// TIA Portal V16 export
// export: Created 2021-11-12T13:32:10.6511653Z, ExportSetting WithDefaults, DisplayName Totally Integrated Automation Portal, DisplayVersion V16 Update 3, DisplayName TIA Portal Version Control Interface, DisplayVersion V16 Update 2, DisplayName TIA Portal Openness, DisplayVersion V16 Update 3, DisplayName SINAMICS Startdrive Advanced, DisplayVersion V16 Update 5, DisplayName SINAMICS Startdrive G130, G150, S120, S150, SINAMICS MV, S210, DisplayVersion V16 Update 5, DisplayName SINAMICS Startdrive G110M, G120, G120C, G120D, G120P, G115D, DisplayVersion V16 Update 5, DisplayName STEP 7 Professional, DisplayVersion V16 Update 3, DisplayName STEP 7 Safety, DisplayVersion V16, DisplayName WinCC UA Professional, DisplayVersion V16 Update 3
DATA_BLOCK "STATUS_180"   // DB2171
{ S7_Optimized_Access := 'TRUE' }
VERSION : 0.1
// stored: AutoNumber false, DBAccessibleFromOPCUA true, IsOnlyStoredInLoadMemory false, IsRetainMemResEnabled false, IsWriteProtectedInAS false, MemoryReserve 100
   VAR
      xxxxx___BinarySensors___xxxxx : Byte;
      xxxxx___BinaryOthers___xxxxx : Byte;
      xxxxx___AnalogueSensors___xxxxx : Byte;
      xxxxx___Drives___xxxxx : Byte;
      xxxxx___MaterialFlow___xxxxx : Byte;
   END_VAR
   VAR RETAIN
      MatCard : Array[1..24, 1..2] of "UDT_MatCard";   // Material card [Line, Pos]
   END_VAR
   VAR
      xxxxx___Other___xxxxx : Byte;
      PartCounter : Int;   // Number of occupied positions in the map
      MapChanged : Bool;   // Map has been changed (pulse)
      xxxxx___SensorAlarms___xxxxx : Byte;
      xxxxx___ProcessAlarms___xxxxx : Byte;
   END_VAR
BEGIN
END_DATA_BLOCK
